# EPICS substitutions: r7FQCRBuilder/iocs/BLTEST-LCH-IOC-01/BLTEST-LCH-IOC-01App/Db/BLTEST-LCH-IOC-01_expanded.substitutions
# This file was automatically generated on Thu 09 May 2019 12:58:43 BST from
# source: /home/jjc62351/work/builderTestBench/r7FQCRBuilder/etc/makeIocs/BLTEST-LCH-IOC-01.xml
#
# *** Please do not edit this file: edit the source file instead. ***
#

# Macros:
#  P             Device Prefix
#  STREAMS_PORT  Stream port
file $(MITSUBISHIROBOT)/db/BARTRobot.db
{
pattern { P, STREAMS_PORT }
    { "BLTEST-LCH-ROBOT-01", "robot_serial" }
}
